# EPICS autosave request: 3-1/GalilSup/Db/galil_reverse_transforms.req
# Reverse transform equations
$(P)$(M)_RTRANSFORMA_SP.VAL
$(P)$(M)_RTRANSFORMB_SP.VAL
$(P)$(M)_RTRANSFORMC_SP.VAL
$(P)$(M)_RTRANSFORMD_SP.VAL
$(P)$(M)_RTRANSFORME_SP.VAL
$(P)$(M)_RTRANSFORMF_SP.VAL
$(P)$(M)_RTRANSFORMG_SP.VAL
$(P)$(M)_RTRANSFORMH_SP.VAL
$(P)$(M)_RTRANSFORMA_SP.DESC
$(P)$(M)_RTRANSFORMB_SP.DESC
$(P)$(M)_RTRANSFORMC_SP.DESC
$(P)$(M)_RTRANSFORMD_SP.DESC
$(P)$(M)_RTRANSFORME_SP.DESC
$(P)$(M)_RTRANSFORMF_SP.DESC
$(P)$(M)_RTRANSFORMG_SP.DESC
$(P)$(M)_RTRANSFORMH_SP.DESC
